(* Logix 5000 project; controller VET 1756-L62 rev 19.52; software revision 19.01; part 15 of 27 *)
(* tags used below, declared in another part *)
   _Eqp : Equipo[800];
   Batch : batch[10];
   dosificador : dosif_struct[20];
   Dosificar_MIC_01 : PHASE;
   Dosificar_MIC_02 : PHASE;
   fecha_plc : DINT;
   hora_plc : DINT;
   SetDInt : DINT[500];
   TabBin : Bins_Setup;
   TabDosif : tabDosif;
   Timer : TIMER[500];
   vdf : VDFS[20];
(* Dosificar_MIC_01, continued *)

ROUTINE Falla   (* ladder *)
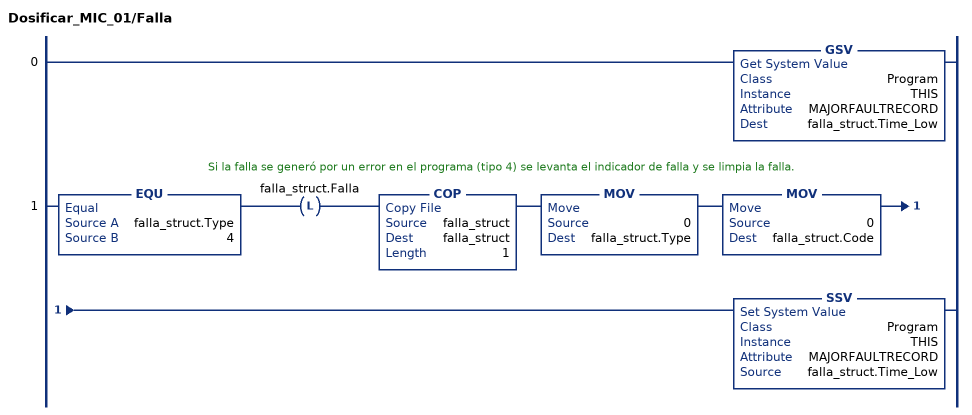
   0: GSV(Program,THIS,MAJORFAULTRECORD,falla_struct.Time_Low);
   // Si la falla se generó por un error en el programa (tipo 4) se levanta el indicador de falla y se limpia la falla.
   1: EQU(falla_struct.Type,4)OTL(falla_struct.Falla)COP(falla_struct,falla_struct,1)MOV(0,falla_struct.Type)MOV(0,falla_struct.Code)SSV(Program,THIS,MAJORFAULTRECORD,falla_struct.Time_Low);
END_ROUTINE

ROUTINE Holding   (* ladder *)
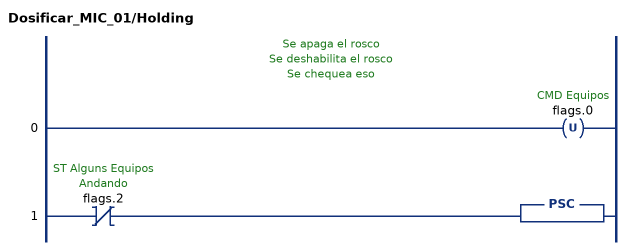
   // Se apaga el rosco
   // Se deshabilita el rosco
   // Se chequea eso
   0: OTU(flags.0);
   1: XIO(flags.2)PSC();
END_ROUTINE

ROUTINE preState   (* ladder *)
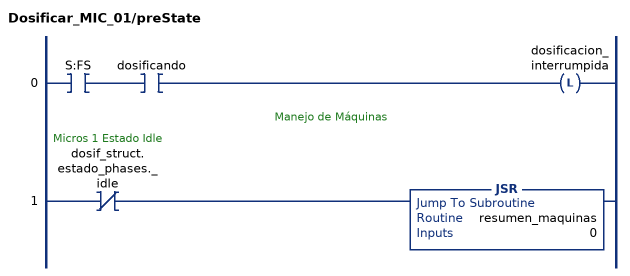
   0: XIC(S:FS)XIC(dosificando)OTL(dosificacion_interrumpida);
   // Manejo de Máquinas
   1: XIO(dosif_struct.estado_phases._idle)JSR(resumen_maquinas,0);
END_ROUTINE

ROUTINE Resetting   (* ladder *)
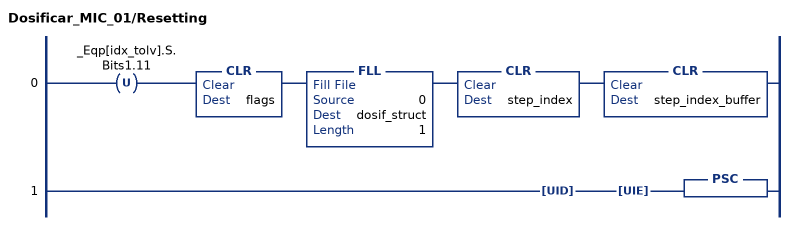
   0: OTU(_Eqp[idx_tolv].S.Bits1.11)CLR(flags)FLL(0,dosif_struct,1)CLR(step_index)CLR(step_index_buffer);
   1: UID()UIE()PSC();
END_ROUTINE

ROUTINE Restarting   (* ladder *)
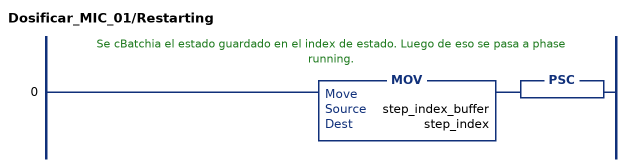
   // Se cBatchia el estado guardado en el index de estado. Luego de eso se pasa a phase running.
   0: MOV(step_index_buffer,step_index)PSC();
END_ROUTINE

ROUTINE resumen_maquinas   (* ladder *)
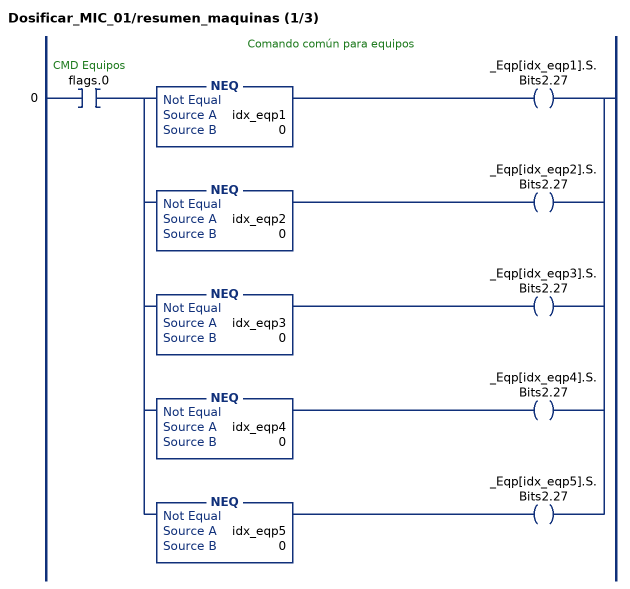
   // Comando común para equipos
   0: XIC(flags.0)[NEQ(idx_eqp1,0) OTE(_Eqp[idx_eqp1].S.Bits2.27) ,NEQ(idx_eqp2,0) OTE(_Eqp[idx_eqp2].S.Bits2.27) ,NEQ(idx_eqp3,0) OTE(_Eqp[idx_eqp3].S.Bits2.27) ,NEQ(idx_eqp4,0) OTE(_Eqp[idx_eqp4].S.Bits2.27) ,NEQ(idx_eqp5,0) OTE(_Eqp[idx_eqp5].S.Bits2.27) ];
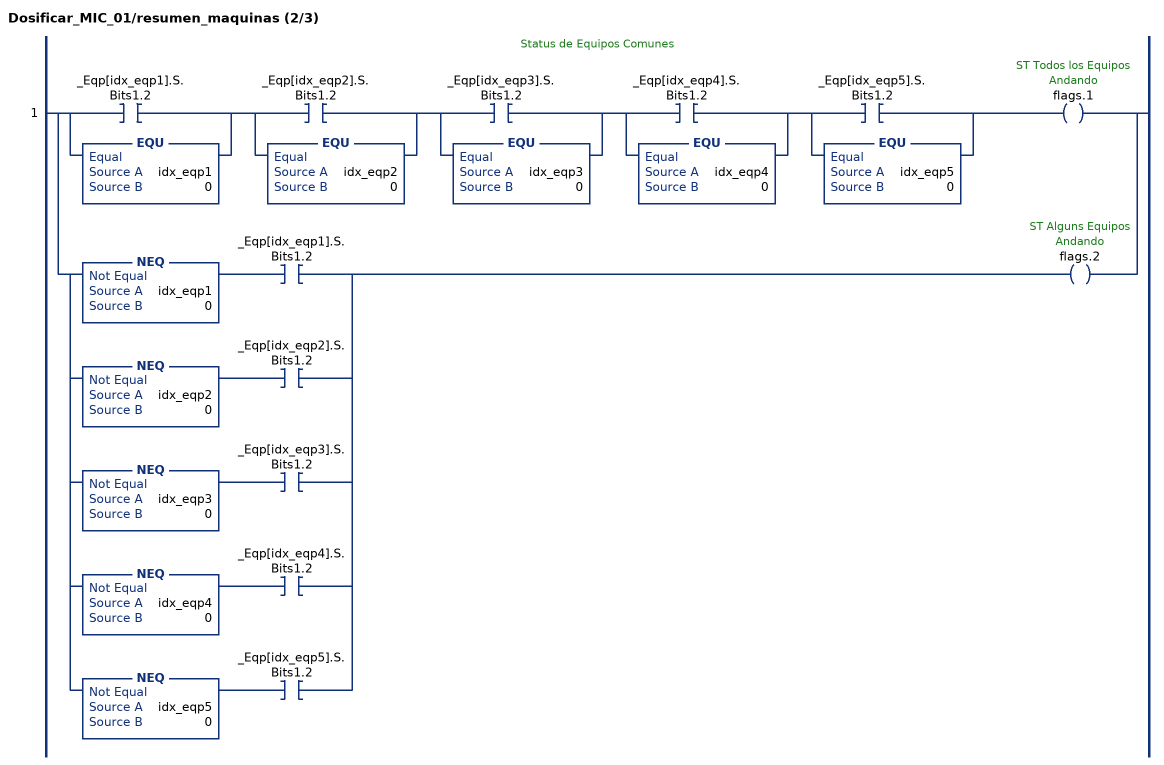
   // Status de Equipos Comunes
   1: [[XIC(_Eqp[idx_eqp1].S.Bits1.2) ,EQU(idx_eqp1,0) ] [XIC(_Eqp[idx_eqp2].S.Bits1.2) ,EQU(idx_eqp2,0) ] [XIC(_Eqp[idx_eqp3].S.Bits1.2) ,EQU(idx_eqp3,0) ] [XIC(_Eqp[idx_eqp4].S.Bits1.2) ,EQU(idx_eqp4,0) ] [XIC(_Eqp[idx_eqp5].S.Bits1.2) ,EQU(idx_eqp5,0) ] OTE(flags.1) ,[NEQ(idx_eqp1,0) XIC(_Eqp[idx_eqp1].S.Bits1.2) ,NEQ(idx_eqp2,0) XIC(_Eqp[idx_eqp2].S.Bits1.2) ,NEQ(idx_eqp3,0) XIC(_Eqp[idx_eqp3].S.Bits1.2) ,NEQ(idx_eqp4,0) XIC(_Eqp[idx_eqp4].S.Bits1.2) ,NEQ(idx_eqp5,0) XIC(_Eqp[idx_eqp5].S.Bits1.2) ] OTE(flags.2) ];
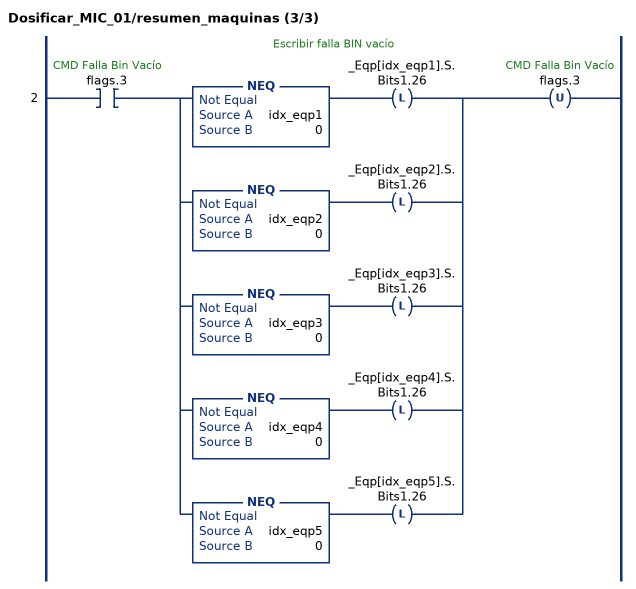
   // Escribir falla BIN vacío
   2: XIC(flags.3)[NEQ(idx_eqp1,0) OTL(_Eqp[idx_eqp1].S.Bits1.26) ,NEQ(idx_eqp2,0) OTL(_Eqp[idx_eqp2].S.Bits1.26) ,NEQ(idx_eqp3,0) OTL(_Eqp[idx_eqp3].S.Bits1.26) ,NEQ(idx_eqp4,0) OTL(_Eqp[idx_eqp4].S.Bits1.26) ,NEQ(idx_eqp5,0) OTL(_Eqp[idx_eqp5].S.Bits1.26) ]OTU(flags.3);
END_ROUTINE

ROUTINE Running   (* ladder *)
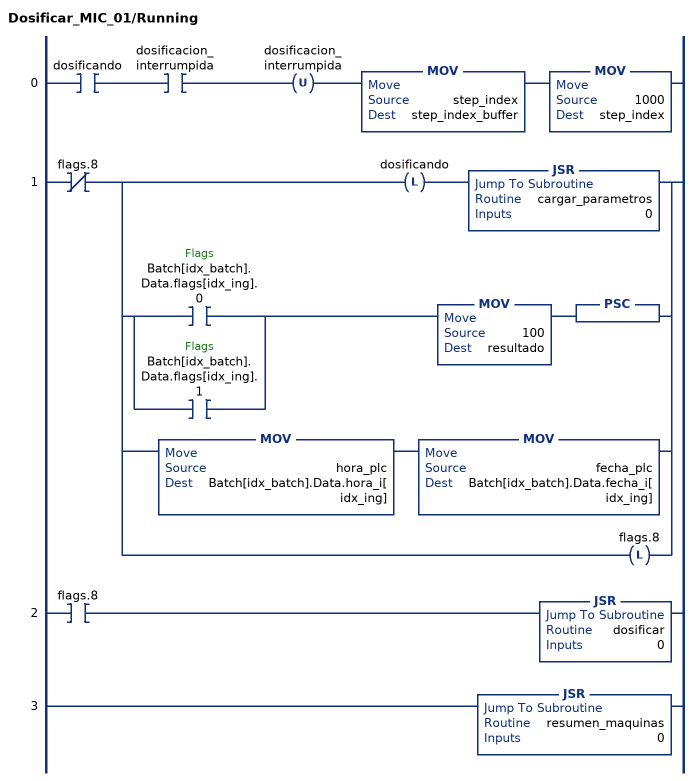
   0: XIC(dosificando)XIC(dosificacion_interrumpida)OTU(dosificacion_interrumpida)MOV(step_index,step_index_buffer)MOV(1000,step_index);
   1: XIO(flags.8)[OTL(dosificando) JSR(cargar_parametros,0) ,[[XIC(Batch[idx_batch].Data.flags[idx_ing].0) ,XIC(Batch[idx_batch].Data.flags[idx_ing].1) ] MOV(100,resultado) PSC() ,MOV(hora_plc,Batch[idx_batch].Data.hora_i[idx_ing]) MOV(fecha_plc,Batch[idx_batch].Data.fecha_i[idx_ing]) ] ,OTL(flags.8) ];
   2: XIC(flags.8)JSR(dosificar,0);
   3: JSR(resumen_maquinas,0);
END_ROUTINE
END_PROGRAM

PROGRAM Dosificar_MIC_02   (* fault routine Falla *)
VAR
   _vel_exp : velocidad_exp := (x := 0.0019866943, curvatura := 1.0, V_inicial := 70.0, V_final := 50.0, V_salida := 50.06262);
   bufferF : REAL[5] := ([0] := 25.010452, [1] := -0.0104522705, [2] := 0.0019866943);
        [2]   // Diferencia entre peso actual y objetivo
   debug : BOOL;
   dosif_extra_ingr : DINT := -1;   // Código del ingrediente que puede ser dosificado extra.
   dosif_struct : ALIAS FOR dosificador[3];
   dosificacion_interrumpida : BOOL;
   dosificando : BOOL;
   error_kg : REAL := 0.1;
   error_per : REAL := 1.25;
   falla_struct : falla_aux;
   flags : DINT;
        .0   // CMD Equipos
        .1   // ST Todos los Equipos Andando
        .2   // ST Alguns Equipos Andando
        .3   // CMD Falla Bin Vacío
        .6   // Bit Precorte
        .7   // Aplicar Precorte
   frq : ALIAS FOR dosif_struct.frq_terreno;
   frq_calculada : REAL := 50.0;
   frq_final : REAL := 50.0;
   frq_inicial : REAL := 70.0;
   hist_precorte : REAL[10] := ([0] := 1.0, [1] := 1.0, [2] := 1.0, [3] := 1.0, [4] := 1.0);
   i_fn : DINT := 17;
   idx_batch : DINT := 3;
   idx_bin : DINT := 31;
   idx_dosif : DINT;   // Índice de dosificador usado
   idx_eqp1 : DINT := 92;
   idx_eqp2 : DINT := 105;
   idx_eqp3 : DINT;
   idx_eqp4 : DINT;
   idx_eqp5 : DINT;
   idx_ing : DINT := 14;
   idx_tabbin : DINT := 1;
   idx_tolv : DINT := 72;   // Índice de Tolva
   limite_err_inf : REAL := 24.9;
   limite_err_sup : REAL := 25.1;
   mensaje : ALIAS FOR dosif_struct.msg;
        .3   // Manual
        .1   // Bin Vacío
        .2   // Predescarga
        .4   // Peso Neto Negativo
        .0   // Error de Pesaje
        .5   // Dosificación interrumpida
   peso_delta : REAL;
   peso_detencion : REAL := 24.951622;
   peso_intermedio : REAL := 12.5;   // Peso límite para dosificación a frecuencia máxima
   peso_max : REAL := 150.0;
   peso_medido : ALIAS FOR dosif_struct.peso_terreno;
   peso_neto : REAL := 25.010452;
   peso_neto_aux : REAL;   // Peso Neto Guardado en caso de Vaciado y llenado de tolva
   peso_objetivo : REAL := 25.0;
   precorte : REAL := 0.050990697;
   respuesta : ALIAS FOR dosif_struct.ans;
        .13   // Peso Neto Cero - Aceptar y Tarar
        .3   // Reintentar Misma Tolva
        .6   // Abortar Ingrediente
        .0   // Aceptar Error
        .10   // Abortar Ingrediente
        .9   // Abortar Batch
        .1   // Abortar Batch
        .2   // Abortar Ingrediente
        .11   // Dosificación Completa
        .5   // Abortar Batch
        .8   // Aceptar Predescarga
        .4   // Cambiar Tolva
        .15   // Abortar Dosificación
        .14   // Continuar Dosificación
        .7   // Pasar a Manual
        .12   // Habilitar Aceptar
        .16   // Abortar Ingrediente
   resultado : ALIAS FOR dosif_struct.resultado;
   return_fn : DINT;
   setD : DINT[5] := ([0] := 1, [1] := 44, [2] := 2, [3] := 1, [4] := 32);
        [1].8   // Con VDF
        [1].0   // Tipo LIW
        [4]   // Destino
        [0]   // Mínima variación de peso para detección de tolva vacía.
        [1].2   // Predescarga
        [1].3   // Aplicar Precorte
        [1].4   // Con Bloqueo de Tolva
        [1].5   // No respeta receta
        [2]   // Mezcladora izquierda
        [3]   // Mezcladora derecha
   setF : REAL[5] := ([0] := 0.1);
        [0]   // Límite para variación de peso
        [1]   // Límite para peso negativo
   step_index : DINT;
   step_index_buffer : DINT;
   T : TIMER[15] := ([0].PRE := 1000, [0].ACC := 240, [0].EN := 1, [0].TT := 1, [1].PRE := 30000, [2].PRE := 3000, [2].ACC := 3039, [2].EN := 1, [2].DN := 1, [3].PRE := 8000, [4].PRE := 1000, [5].PRE := 1000, [6].PRE := 1000, [7].PRE := 2500, [8].PRE := 1000, [9].PRE := 1000, [10].PRE := 5000);
   t_espera : DINT := 3000;
   t_pulso : DINT := 6000;
   tara : REAL := 115.98935;
   v : DINT;
END_VAR

ROUTINE _fn_dividir_ingrediente   (* ladder *)
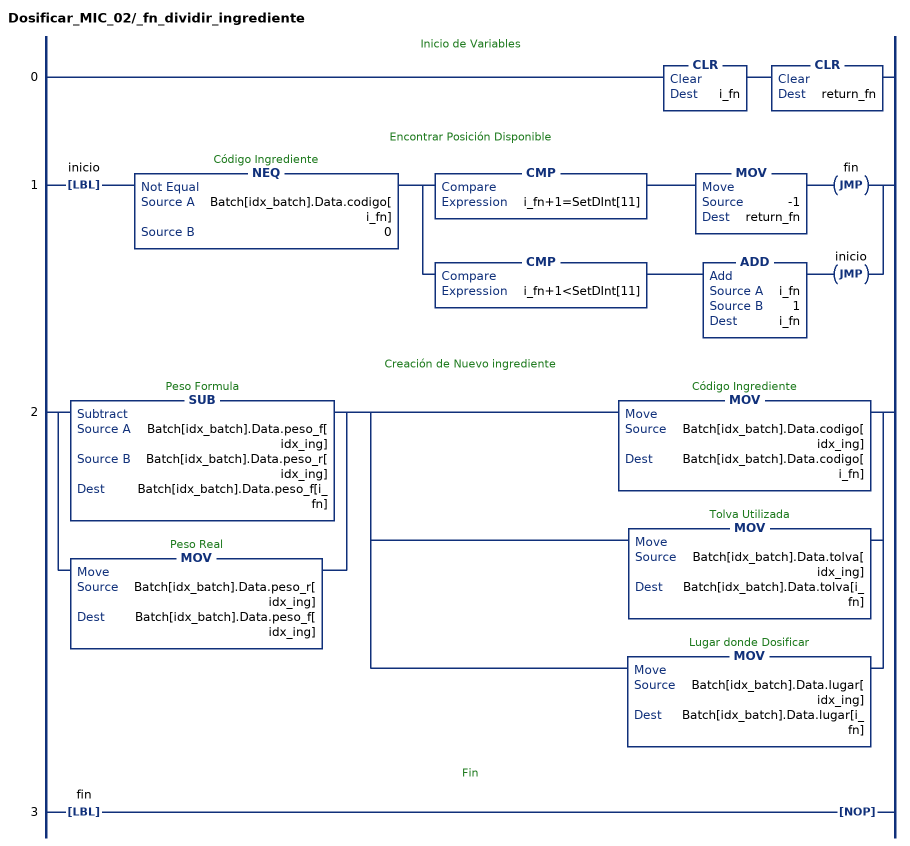
   // Inicio de Variables
   0: CLR(i_fn)CLR(return_fn);
   // Encontrar Posición Disponible
   1: LBL(inicio)NEQ(Batch[idx_batch].Data.codigo[i_fn],0)[CMP(i_fn+1=SetDInt[11]) MOV(-1,return_fn) JMP(fin) ,CMP(i_fn+1<SetDInt[11]) ADD(i_fn,1,i_fn) JMP(inicio) ];
   // Creación de Nuevo ingrediente
   2: [SUB(Batch[idx_batch].Data.peso_f[idx_ing],Batch[idx_batch].Data.peso_r[idx_ing],Batch[idx_batch].Data.peso_f[i_fn]) ,MOV(Batch[idx_batch].Data.peso_r[idx_ing],Batch[idx_batch].Data.peso_f[idx_ing]) ][MOV(Batch[idx_batch].Data.codigo[idx_ing],Batch[idx_batch].Data.codigo[i_fn]) ,MOV(Batch[idx_batch].Data.tolva[idx_ing],Batch[idx_batch].Data.tolva[i_fn]) ,MOV(Batch[idx_batch].Data.lugar[idx_ing],Batch[idx_batch].Data.lugar[i_fn]) ];
   // Fin
   3: LBL(fin)NOP();
END_ROUTINE

ROUTINE Aborting   (* ladder *)
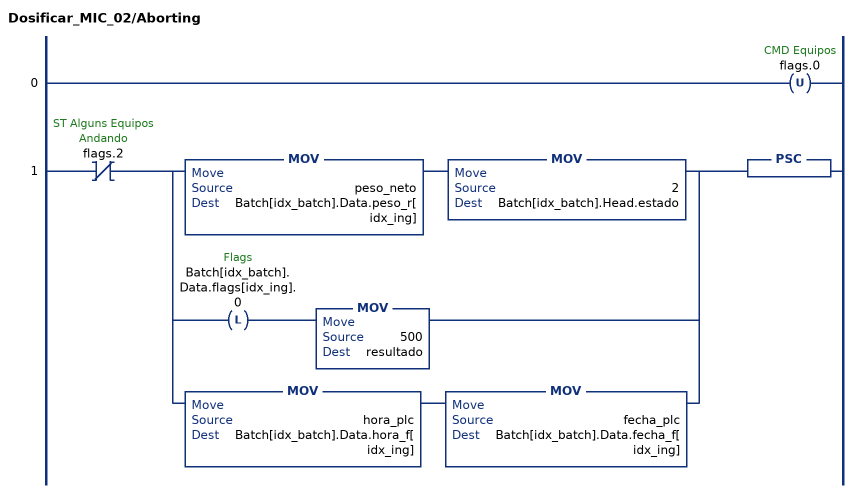
   0: OTU(flags.0);
   1: XIO(flags.2)[MOV(peso_neto,Batch[idx_batch].Data.peso_r[idx_ing]) MOV(2,Batch[idx_batch].Head.estado) ,OTL(Batch[idx_batch].Data.flags[idx_ing].0) MOV(500,resultado) ,MOV(hora_plc,Batch[idx_batch].Data.hora_f[idx_ing]) MOV(fecha_plc,Batch[idx_batch].Data.fecha_f[idx_ing]) ]PSC();
END_ROUTINE

ROUTINE calculo_frecuencia   (* ladder *)
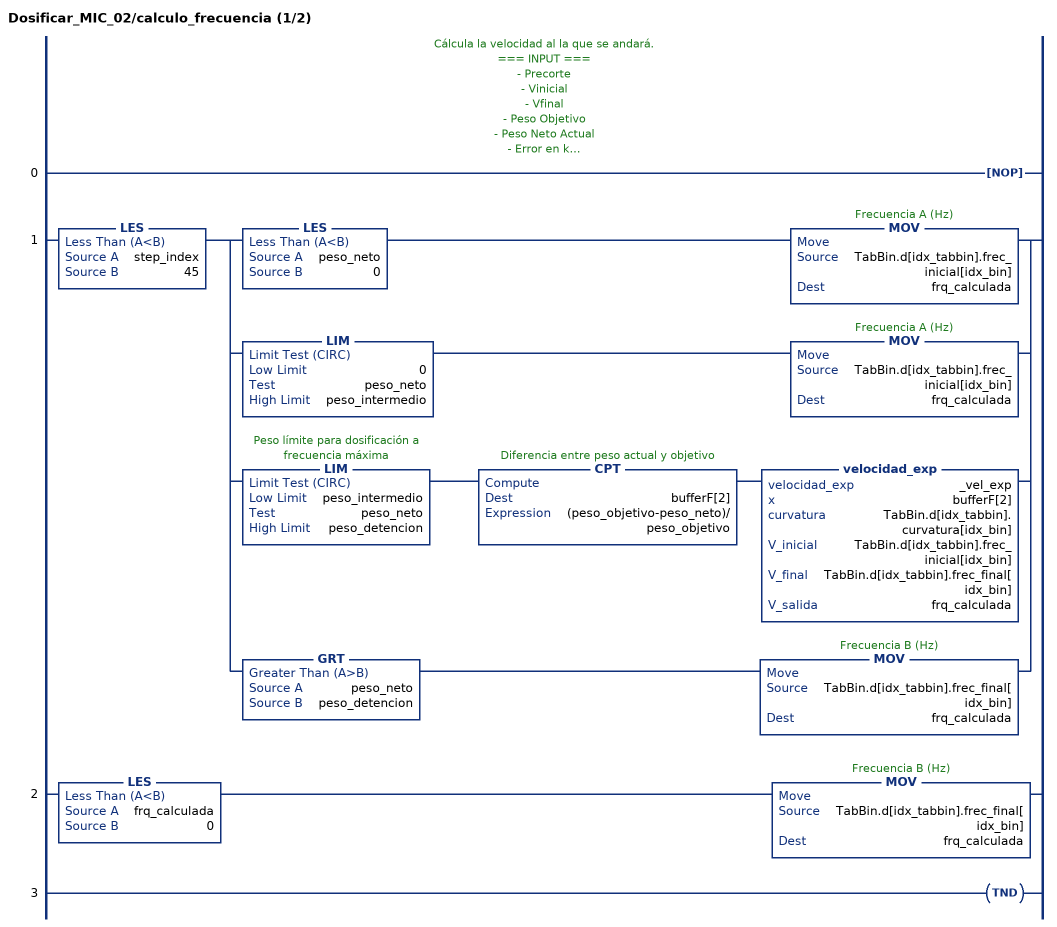
   // Cálcula la velocidad al la que se andará.
   // === INPUT ===
   // - Precorte
   // - Vinicial
   // - Vfinal
   // - Peso Objetivo
   // - Peso Neto Actual
   // - Error en kg
   // === OUTPUT ===
   // - Vactual
   0: NOP();
   1: LES(step_index,45)[LES(peso_neto,0) MOV(TabBin.d[idx_tabbin].frec_inicial[idx_bin],frq_calculada) ,LIM(0,peso_neto,peso_intermedio) MOV(TabBin.d[idx_tabbin].frec_inicial[idx_bin],frq_calculada) ,LIM(peso_intermedio,peso_neto,peso_detencion) CPT(bufferF[2],(peso_objetivo-peso_neto)/peso_objetivo) velocidad_exp(_vel_exp,bufferF[2],TabBin.d[idx_tabbin].curvatura[idx_bin],TabBin.d[idx_tabbin].frec_inicial[idx_bin],TabBin.d[idx_tabbin].frec_final[idx_bin],frq_calculada) ,GRT(peso_neto,peso_detencion) MOV(TabBin.d[idx_tabbin].frec_final[idx_bin],frq_calculada) ];
   2: LES(frq_calculada,0)MOV(TabBin.d[idx_tabbin].frec_final[idx_bin],frq_calculada);
   3: TND();
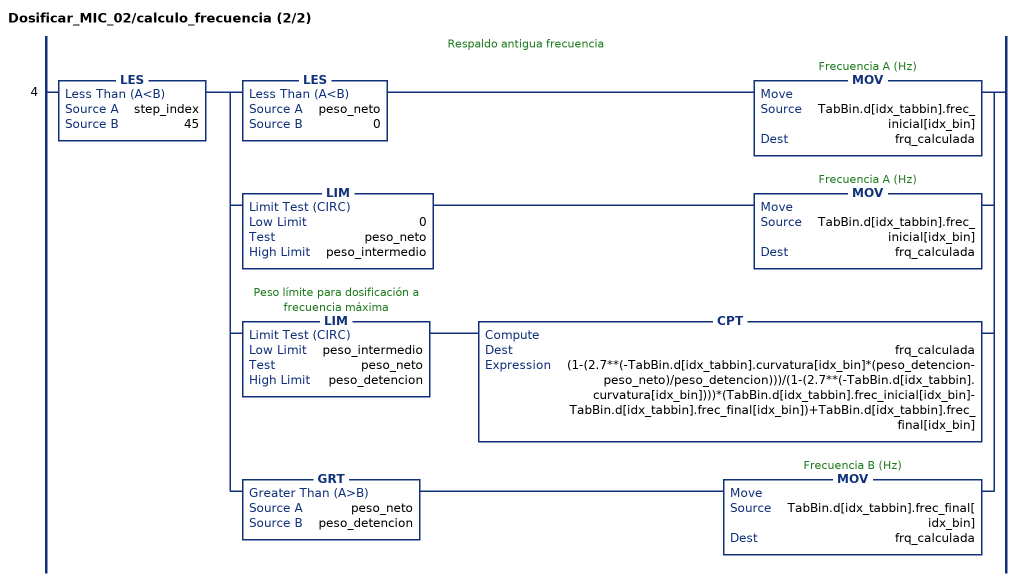
   // Respaldo antigua frecuencia
   4: LES(step_index,45)[LES(peso_neto,0) MOV(TabBin.d[idx_tabbin].frec_inicial[idx_bin],frq_calculada) ,LIM(0,peso_neto,peso_intermedio) MOV(TabBin.d[idx_tabbin].frec_inicial[idx_bin],frq_calculada) ,LIM(peso_intermedio,peso_neto,peso_detencion) CPT(frq_calculada,(1-(2.7**(-TabBin.d[idx_tabbin].curvatura[idx_bin]*(peso_detencion-peso_neto)/peso_detencion)))/(1-(2.7**(-TabBin.d[idx_tabbin].curvatura[idx_bin])))*(TabBin.d[idx_tabbin].frec_inicial[idx_bin]-TabBin.d[idx_tabbin].frec_final[idx_bin])+TabBin.d[idx_tabbin].frec_final[idx_bin]) ,GRT(peso_neto,peso_detencion) MOV(TabBin.d[idx_tabbin].frec_final[idx_bin],frq_calculada) ];
END_ROUTINE

ROUTINE cargar_parametros   (* ladder *)
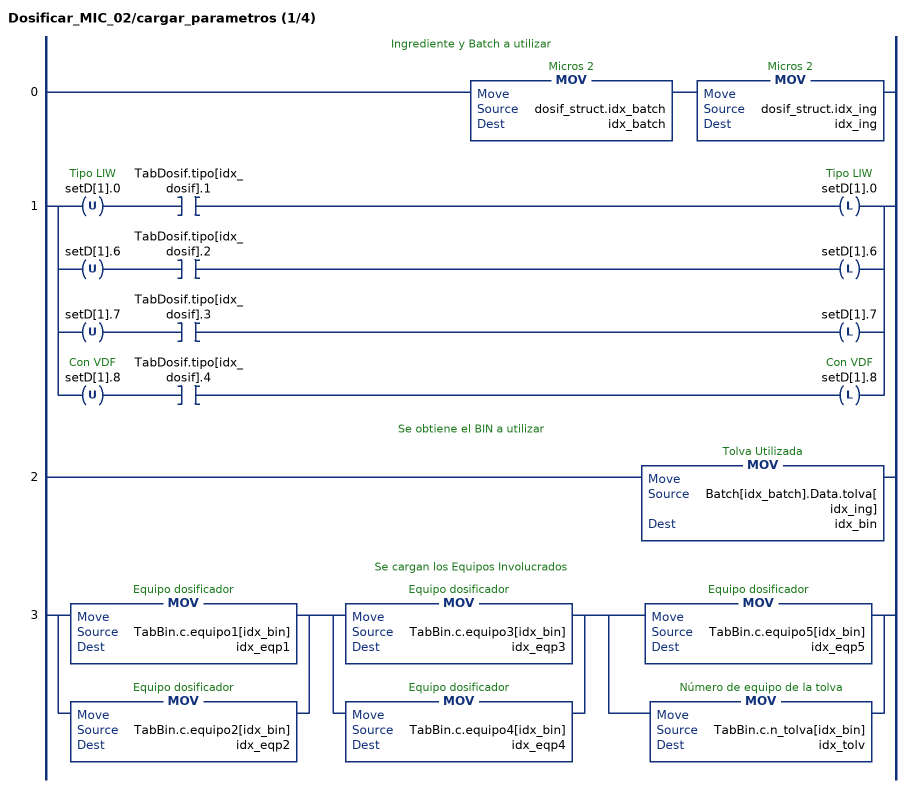
   // Ingrediente y Batch a utilizar
   0: MOV(dosif_struct.idx_batch,idx_batch)MOV(dosif_struct.idx_ing,idx_ing);
   1: [OTU(setD[1].0) XIC(TabDosif.tipo[idx_dosif].1) OTL(setD[1].0) ,OTU(setD[1].6) XIC(TabDosif.tipo[idx_dosif].2) OTL(setD[1].6) ,OTU(setD[1].7) XIC(TabDosif.tipo[idx_dosif].3) OTL(setD[1].7) ,OTU(setD[1].8) XIC(TabDosif.tipo[idx_dosif].4) OTL(setD[1].8) ];
   // Se obtiene el BIN a utilizar
   2: MOV(Batch[idx_batch].Data.tolva[idx_ing],idx_bin);
   // Se cargan los Equipos Involucrados
   3: [MOV(TabBin.c.equipo1[idx_bin],idx_eqp1) ,MOV(TabBin.c.equipo2[idx_bin],idx_eqp2) ][MOV(TabBin.c.equipo3[idx_bin],idx_eqp3) ,MOV(TabBin.c.equipo4[idx_bin],idx_eqp4) ][MOV(TabBin.c.equipo5[idx_bin],idx_eqp5) ,MOV(TabBin.c.n_tolva[idx_bin],idx_tolv) ];
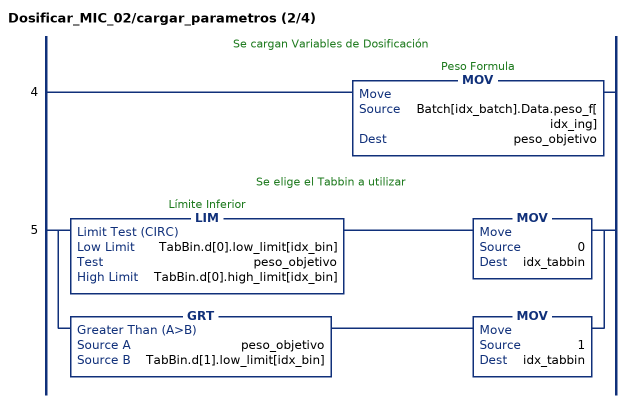
   // Se cargan Variables de Dosificación
   4: MOV(Batch[idx_batch].Data.peso_f[idx_ing],peso_objetivo);
   // Se elige el Tabbin a utilizar
   5: [LIM(TabBin.d[0].low_limit[idx_bin],peso_objetivo,TabBin.d[0].high_limit[idx_bin]) MOV(0,idx_tabbin) ,GRT(peso_objetivo,TabBin.d[1].low_limit[idx_bin]) MOV(1,idx_tabbin) ];
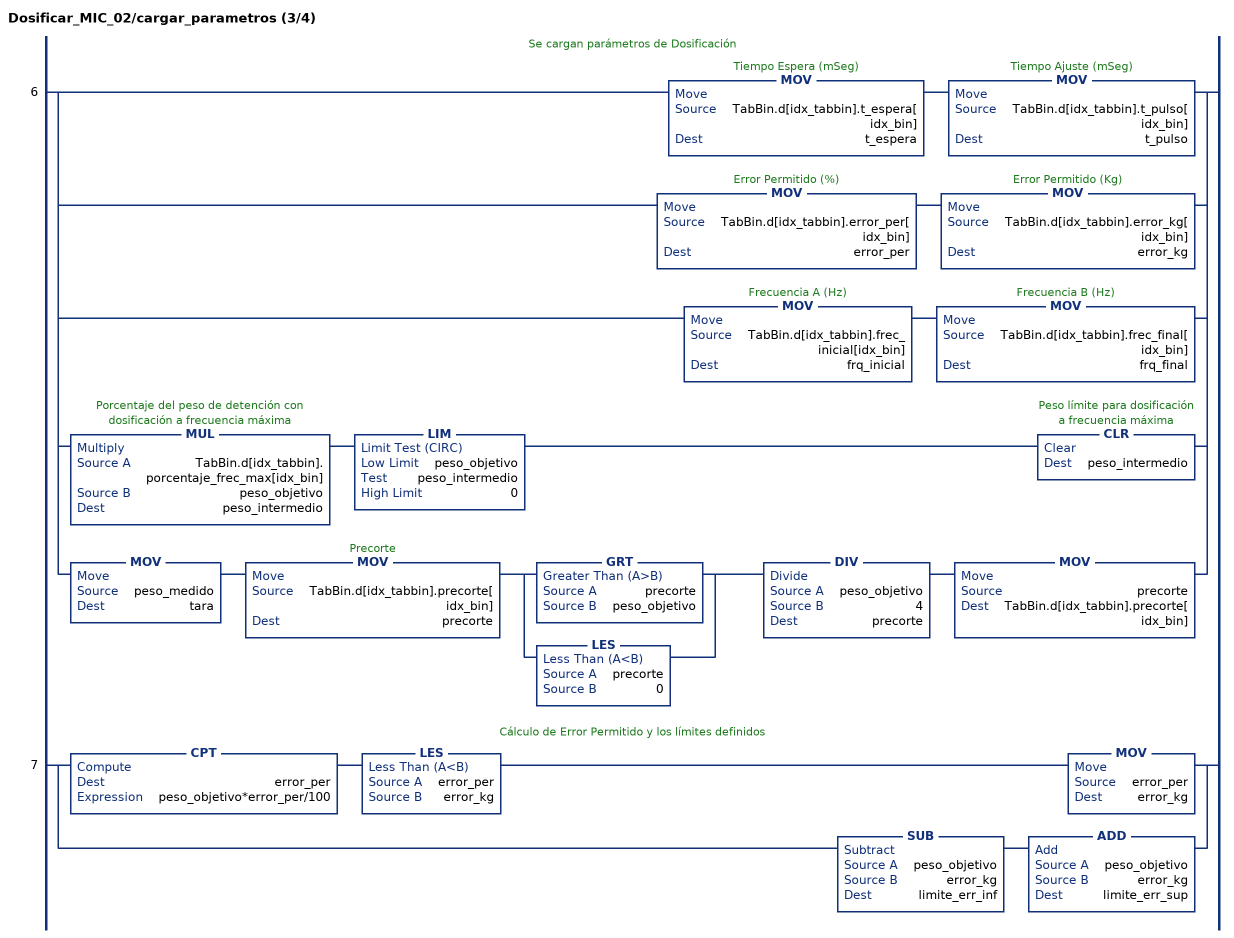
   // Se cargan parámetros de Dosificación
   6: [MOV(TabBin.d[idx_tabbin].t_espera[idx_bin],t_espera) MOV(TabBin.d[idx_tabbin].t_pulso[idx_bin],t_pulso) ,MOV(TabBin.d[idx_tabbin].error_per[idx_bin],error_per) MOV(TabBin.d[idx_tabbin].error_kg[idx_bin],error_kg) ,MOV(TabBin.d[idx_tabbin].frec_inicial[idx_bin],frq_inicial) MOV(TabBin.d[idx_tabbin].frec_final[idx_bin],frq_final) ,MUL(TabBin.d[idx_tabbin].porcentaje_frec_max[idx_bin],peso_objetivo,peso_intermedio) LIM(peso_objetivo,peso_intermedio,0) CLR(peso_intermedio) ,MOV(peso_medido,tara) MOV(TabBin.d[idx_tabbin].precorte[idx_bin],precorte) [GRT(precorte,peso_objetivo) ,LES(precorte,0) ] DIV(peso_objetivo,4,precorte) MOV(precorte,TabBin.d[idx_tabbin].precorte[idx_bin]) ];
   // Cálculo de Error Permitido y los límites definidos
   7: [CPT(error_per,peso_objetivo*error_per/100) LES(error_per,error_kg) MOV(error_per,error_kg) ,SUB(peso_objetivo,error_kg,limite_err_inf) ADD(peso_objetivo,error_kg,limite_err_sup) ];
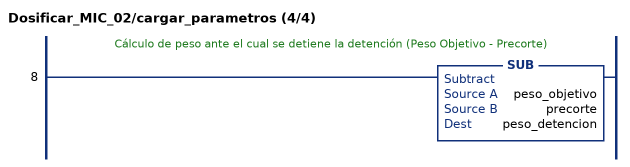
   // Cálculo de peso ante el cual se detiene la detención (Peso Objetivo - Precorte)
   8: SUB(peso_objetivo,precorte,peso_detencion);
END_ROUTINE

ROUTINE dosificar   (* ladder *)
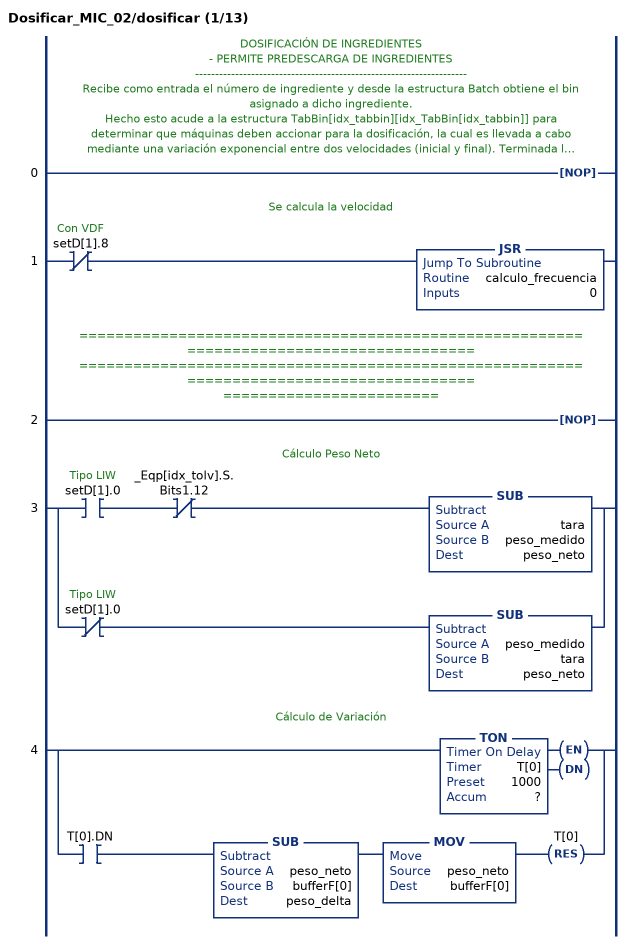
   // DOSIFICACIÓN DE INGREDIENTES
   // - PERMITE PREDESCARGA DE INGREDIENTES
   // --------------------------------------------------------------------
   // Recibe como entrada el número de ingrediente y desde la estructura Batch obtiene el bin asignado a dicho ingrediente.
   // Hecho esto acude a la estructura TabBin[idx_tabbin][idx_TabBin[idx_tabbin]] para determinar que máquinas deben accionar para la dosificación, la cual es llevada a cabo
   // mediante una variación exponencial entre dos velocidades (inicial y final). Terminada la dosificación, se retornan o consolidan los aprendizajes
   // prBatchios de la dosificación, reflejados en un precorte ajustado.
   0: NOP();
   // Se calcula la velocidad
   1: XIO(setD[1].8)JSR(calculo_frecuencia,0);
   // ========================================================================================
   // ========================================================================================
   // ========================
   2: NOP();
   // Cálculo Peso Neto
   3: [XIC(setD[1].0) XIO(_Eqp[idx_tolv].S.Bits1.12) SUB(tara,peso_medido,peso_neto) ,XIO(setD[1].0) SUB(peso_medido,tara,peso_neto) ];
   // Cálculo de Variación
   4: [TON(T[0],?,?) ,XIC(T[0].DN) SUB(peso_neto,bufferF[0],peso_delta) MOV(peso_neto,bufferF[0]) RES(T[0]) ];
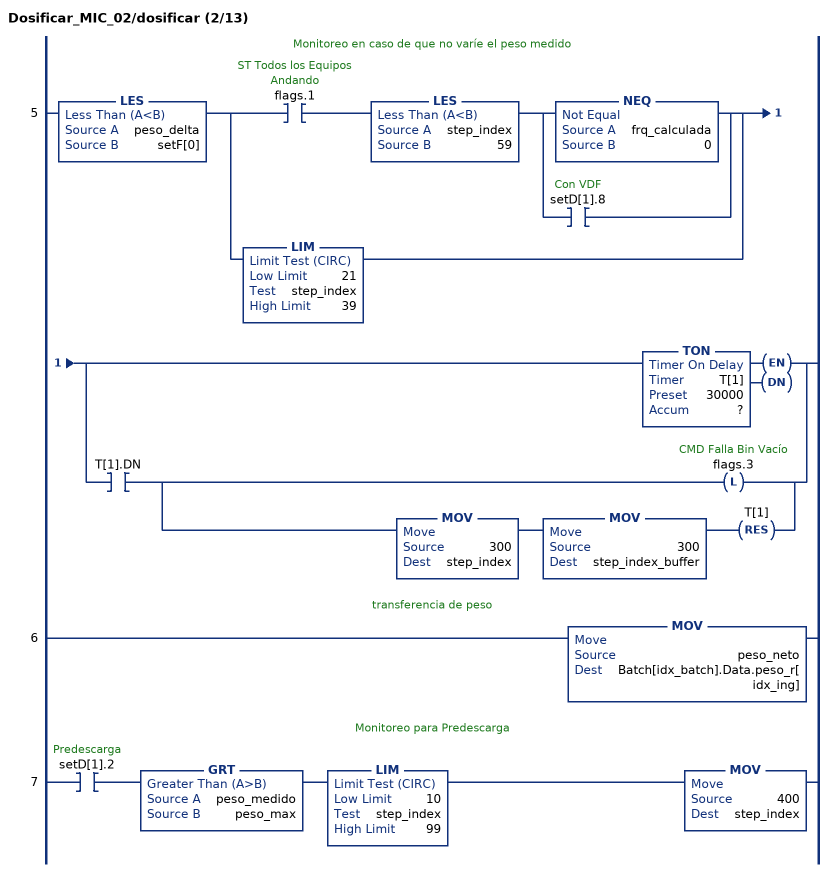
   // Monitoreo en caso de que no varíe el peso medido
   5: LES(peso_delta,setF[0])[XIC(flags.1) LES(step_index,59) [NEQ(frq_calculada,0) ,XIC(setD[1].8) ] ,LIM(21,step_index,39) ][TON(T[1],?,?) ,XIC(T[1].DN) [OTL(flags.3) ,MOV(300,step_index) MOV(300,step_index_buffer) RES(T[1]) ] ];
   // transferencia de peso
   6: MOV(peso_neto,Batch[idx_batch].Data.peso_r[idx_ing]);
   // Monitoreo para Predescarga
   7: XIC(setD[1].2)GRT(peso_medido,peso_max)LIM(10,step_index,99)MOV(400,step_index);
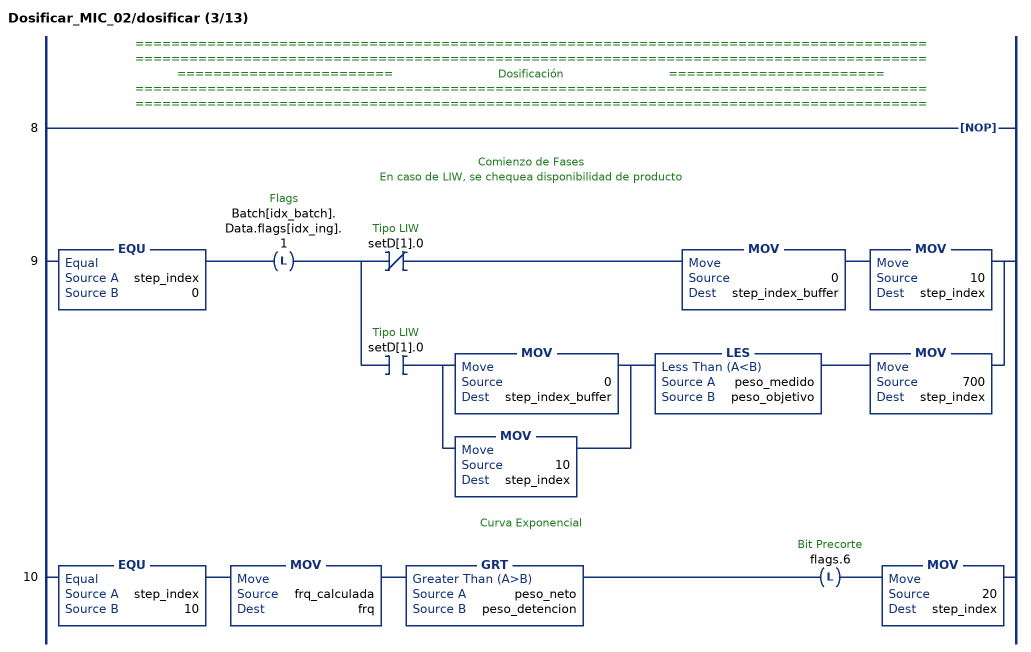
   // ========================================================================================
   // ========================================================================================
   // ========================                              Dosificación                              ========================
   // ========================================================================================
   // ========================================================================================
   8: NOP();
   // Comienzo de Fases
   // En caso de LIW, se chequea disponibilidad de producto
   9: EQU(step_index,0)OTL(Batch[idx_batch].Data.flags[idx_ing].1)[XIO(setD[1].0) MOV(0,step_index_buffer) MOV(10,step_index) ,XIC(setD[1].0) [MOV(0,step_index_buffer) ,MOV(10,step_index) ] LES(peso_medido,peso_objetivo) MOV(700,step_index) ];
   // Curva Exponencial
   10: EQU(step_index,10)MOV(frq_calculada,frq)GRT(peso_neto,peso_detencion)OTL(flags.6)MOV(20,step_index);
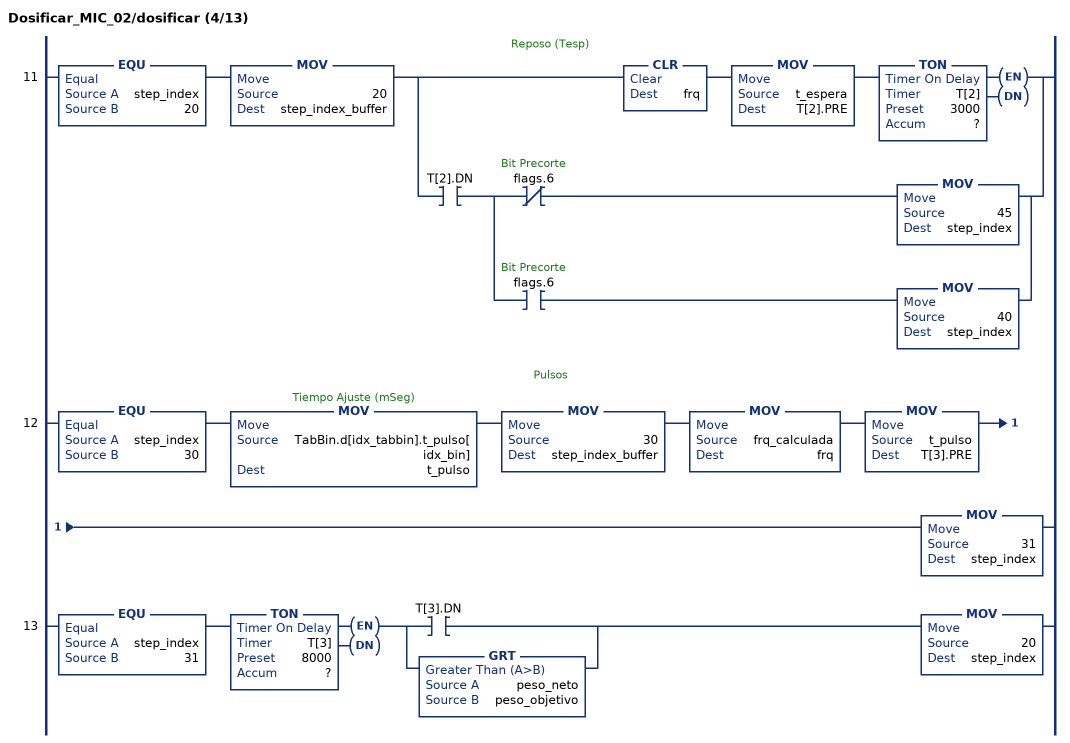
   // Reposo (Tesp)
   11: EQU(step_index,20)MOV(20,step_index_buffer)[CLR(frq) MOV(t_espera,T[2].PRE) TON(T[2],?,?) ,XIC(T[2].DN) [XIO(flags.6) MOV(45,step_index) ,XIC(flags.6) MOV(40,step_index) ] ];
   // Pulsos
   12: EQU(step_index,30)MOV(TabBin.d[idx_tabbin].t_pulso[idx_bin],t_pulso)MOV(30,step_index_buffer)MOV(frq_calculada,frq)MOV(t_pulso,T[3].PRE)MOV(31,step_index);
   13: EQU(step_index,31)TON(T[3],?,?)[XIC(T[3].DN) ,GRT(peso_neto,peso_objetivo) ]MOV(20,step_index);
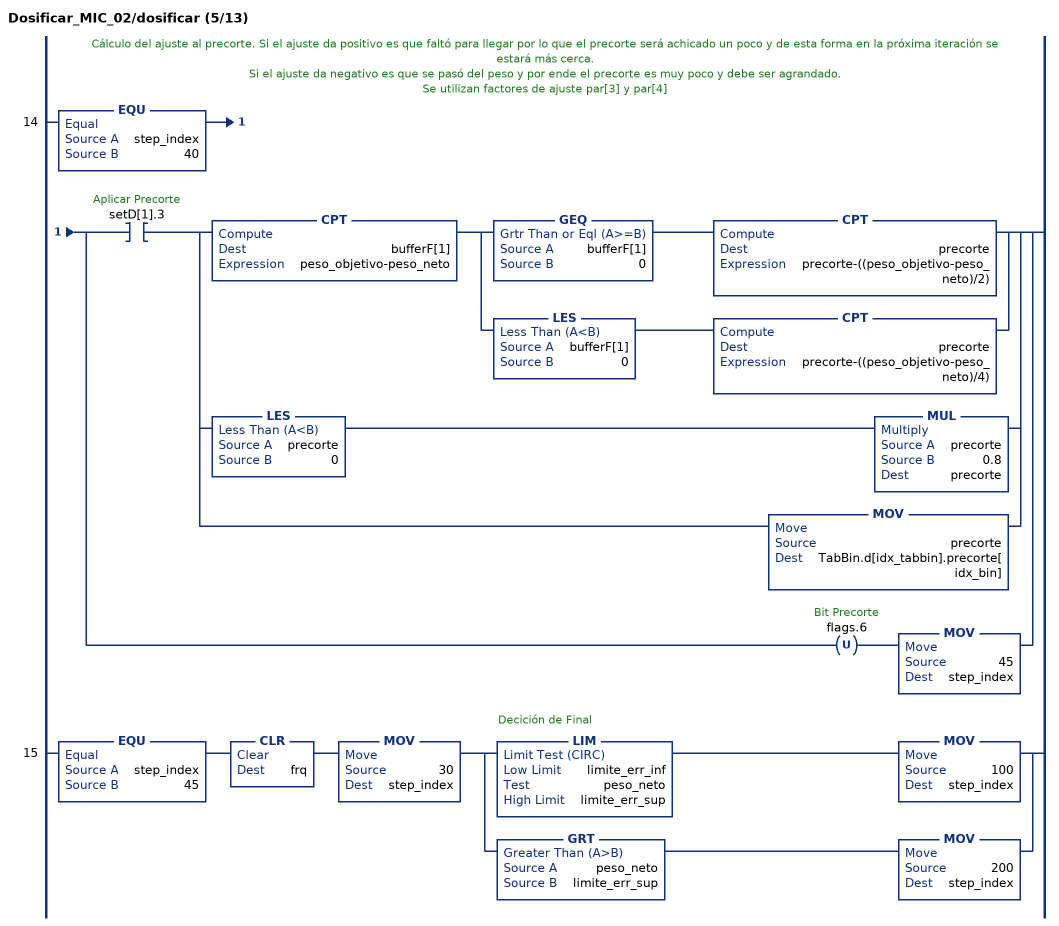
   // Cálculo del ajuste al precorte. Si el ajuste da positivo es que faltó para llegar por lo que el precorte será achicado un poco y de esta forma en la próxima iteración se estará más cerca.
   // Si el ajuste da negativo es que se pasó del peso y por ende el precorte es muy poco y debe ser agrandado.
   // Se utilizan factores de ajuste par[3] y par[4]
   14: EQU(step_index,40)[XIC(setD[1].3) [CPT(bufferF[1],peso_objetivo-peso_neto) [GEQ(bufferF[1],0) CPT(precorte,precorte-((peso_objetivo-peso_neto)/2)) ,LES(bufferF[1],0) CPT(precorte,precorte-((peso_objetivo-peso_neto)/4)) ] ,LES(precorte,0) MUL(precorte,0.8,precorte) ,MOV(precorte,TabBin.d[idx_tabbin].precorte[idx_bin]) ] ,OTU(flags.6) MOV(45,step_index) ];
   // Decición de Final
   15: EQU(step_index,45)CLR(frq)MOV(30,step_index)[LIM(limite_err_inf,peso_neto,limite_err_sup) MOV(100,step_index) ,GRT(peso_neto,limite_err_sup) MOV(200,step_index) ];
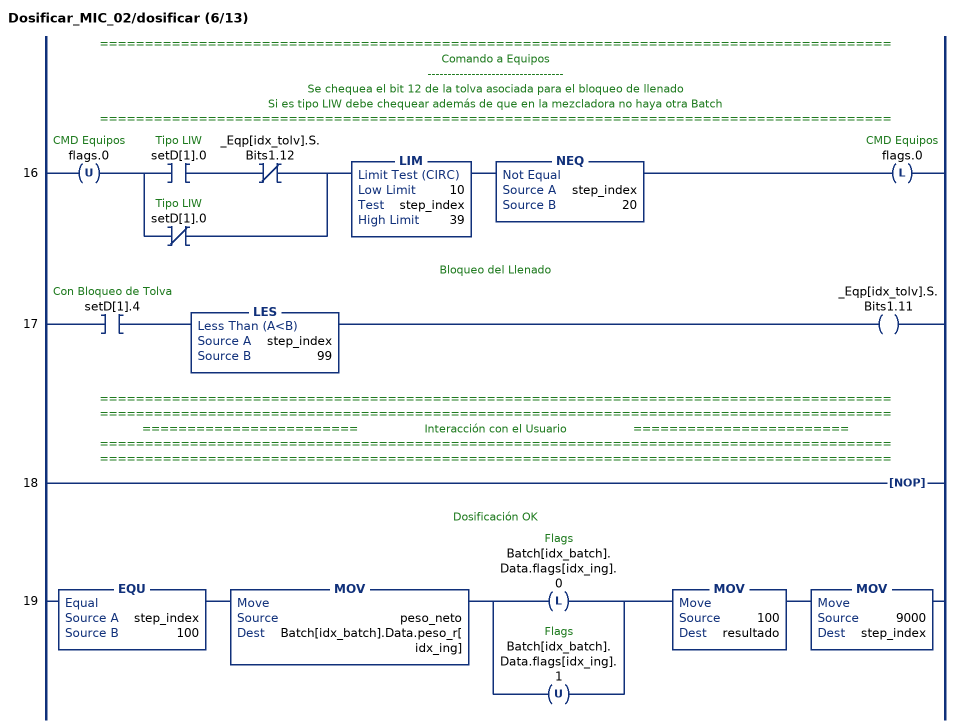
   // ========================================================================================
   // Comando a Equipos
   // ----------------------------------
   // Se chequea el bit 12 de la tolva asociada para el bloqueo de llenado
   // Si es tipo LIW debe chequear además de que en la mezcladora no haya otra Batch
   // ========================================================================================
   16: OTU(flags.0)[XIC(setD[1].0) XIO(_Eqp[idx_tolv].S.Bits1.12) ,XIO(setD[1].0) ]LIM(10,step_index,39)NEQ(step_index,20)OTL(flags.0);
   // Bloqueo del Llenado
   17: XIC(setD[1].4)LES(step_index,99)OTE(_Eqp[idx_tolv].S.Bits1.11);
   // ========================================================================================
   // ========================================================================================
   // ========================                   Interacción con el Usuario                   ========================
   // ========================================================================================
   // ========================================================================================
   18: NOP();
   // Dosificación OK
   19: EQU(step_index,100)MOV(peso_neto,Batch[idx_batch].Data.peso_r[idx_ing])[OTL(Batch[idx_batch].Data.flags[idx_ing].0) ,OTU(Batch[idx_batch].Data.flags[idx_ing].1) ]MOV(100,resultado)MOV(9000,step_index);
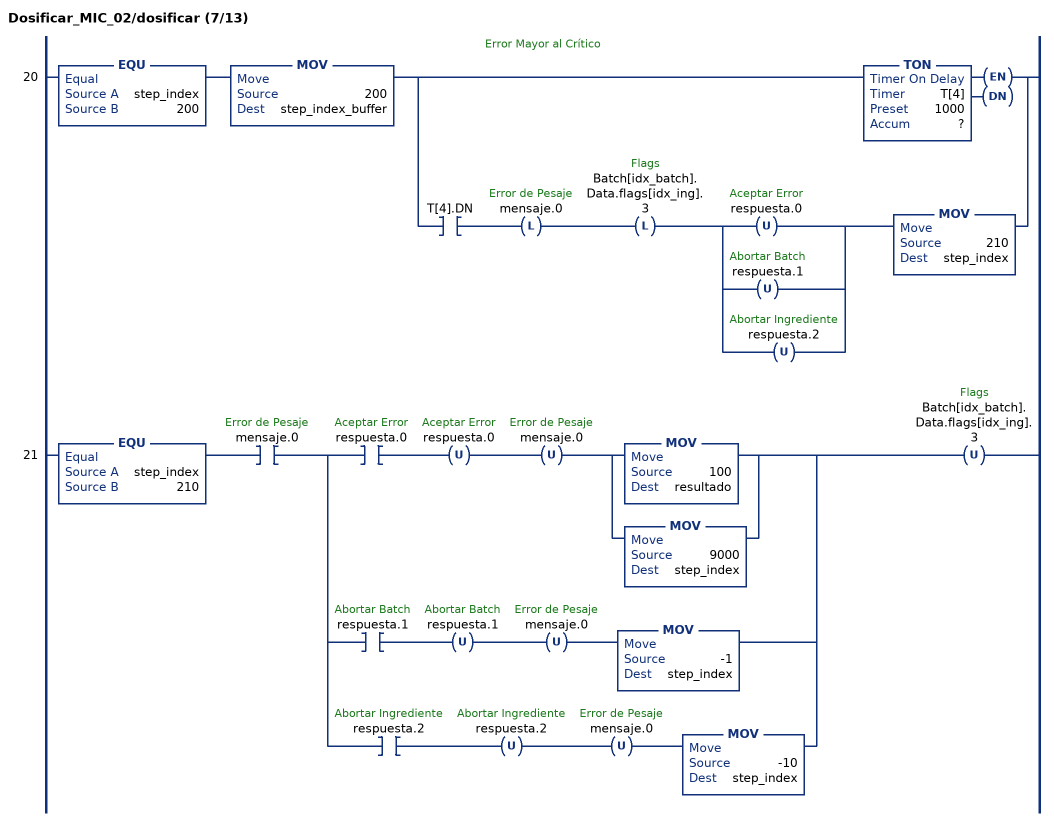
   // Error Mayor al Crítico
   20: EQU(step_index,200)MOV(200,step_index_buffer)[TON(T[4],?,?) ,XIC(T[4].DN) OTL(mensaje.0) OTL(Batch[idx_batch].Data.flags[idx_ing].3) [OTU(respuesta.0) ,OTU(respuesta.1) ,OTU(respuesta.2) ] MOV(210,step_index) ];
   21: EQU(step_index,210)XIC(mensaje.0)[XIC(respuesta.0) OTU(respuesta.0) OTU(mensaje.0) [MOV(100,resultado) ,MOV(9000,step_index) ] ,XIC(respuesta.1) OTU(respuesta.1) OTU(mensaje.0) MOV(-1,step_index) ,XIC(respuesta.2) OTU(respuesta.2) OTU(mensaje.0) MOV(-10,step_index) ]OTU(Batch[idx_batch].Data.flags[idx_ing].3);
